// Block: PAC_320_Data

DATA_BLOCK PAC_320_Data
VERSION : 0.1
   NON_RETAIN
   VAR
      ActualData : udt_PAC3220;
      MES_MeasuringItem : DInt;
      MES_TotalActiveEnergy : LReal;
      MES_60sActiveEnergy : LReal;
      TimeStamp : DTL;
      Aux : Struct
         MinTimer : IEC_TIMER;
         MinutePulse : Bool;
      END_STRUCT;
   END_VAR

BEGIN
   // No initialization required
END_DATA_BLOCK
